// TIA Portal project "2022.10.18_视觉功能块（FB）" (V17)

(* hardware
DEVICE "S7-1200 station_1"  S7-1200 Station
   slot 0: "Rack_0"  S7-1200 Rack  Rack  V1.0
   slot 1: "PLC_1"  CPU 1215C DC/DC/Rly  6ES7 215-1HG40-0XB0  V4.5
*)

// ===== PLC "PLC_1"  CPU 1215C DC/DC/Rly =====

VAR_GLOBAL   // PLC tag table "默认变量表"
   "生成随机数" AT %M10.0 : Bool;
   "Tag_1" AT %M10.1 : Bool;
   "Tag_2" AT %M10.2 : Bool;
END_VAR

DATA_BLOCK "队列操作_DB"   // DB1
{ S7_Optimized_Access := 'TRUE' }
VERSION : 0.1
// stored: InstanceOfName 队列操作
"队列操作"
BEGIN
END_DATA_BLOCK

FUNCTION_BLOCK "队列操作"   // FB1, LAD
{ S7_Optimized_Access := 'TRUE' }
VERSION : 0.1
   VAR_INPUT
      生成随机数 : Bool;
      写入队列 : Bool;
      踢出队列 : Bool;
   END_VAR
   VAR_OUTPUT
      待加入队列的值 : UDInt;
      待踢出的数值 : UDInt;
   END_VAR
   VAR
      队列数据 : Array[1..10] of UDInt;
      数据暂存区 : Array[1..10] of UDInt;
      上一个RLO值1 : Bool;
      上一个RLO值2 : Bool;
      上一个RLO值3 : Bool;
      INDEX : DInt;
      RET_VAL : Int;
      系统时间 : DTL;
   END_VAR
   VAR_TEMP   // added for the SCL form of the ladder/FBD networks
      _w1 : Bool;
   END_VAR
BEGIN

REGION Network 1: 生成一个随机数
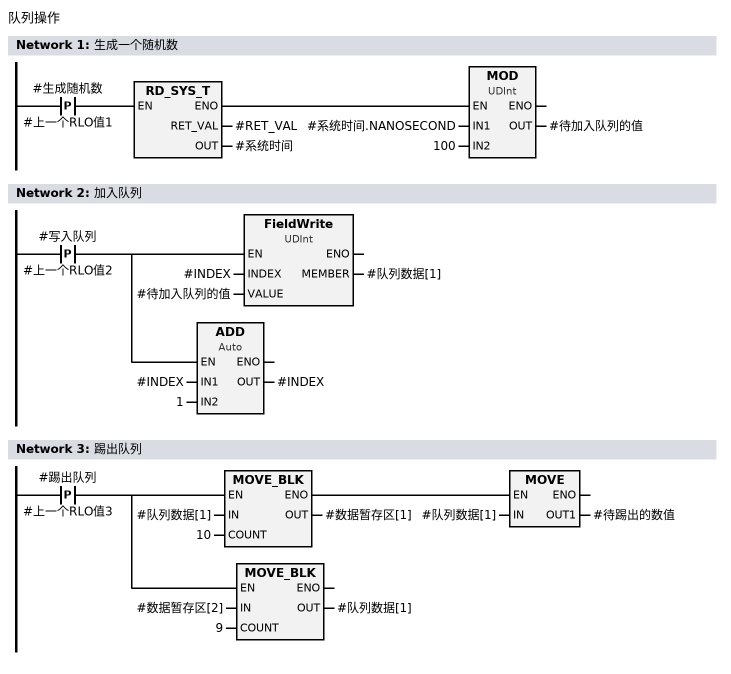
   // ENO of a box is taken as its EN; it also drops when the box reports an error
   #_w1 := #生成随机数 AND NOT #上一个RLO值1;   // rising edge of #生成随机数
   #上一个RLO值1 := #生成随机数;
   IF #_w1 THEN
       #RET_VAL := RD_SYS_T(OUT => #系统时间);
       #待加入队列的值 := #系统时间.NANOSECOND MOD 100;
   END_IF;
END_REGION

REGION Network 2: 加入队列
   // no SCL statement known for FieldWrite: written as a call
   #_w1 := #写入队列 AND NOT #上一个RLO值2;   // rising edge of #写入队列
   #上一个RLO值2 := #写入队列;
   IF #_w1 THEN
       FieldWrite(index := #INDEX, value := #待加入队列的值, member => #队列数据[1]);
       #INDEX := #INDEX + 1;
   END_IF;
END_REGION

REGION Network 3: 踢出队列
   #_w1 := #踢出队列 AND NOT #上一个RLO值3;   // rising edge of #踢出队列
   #上一个RLO值3 := #踢出队列;
   IF #_w1 THEN
       MOVE_BLK(IN := #队列数据[1], COUNT := 10, OUT => #数据暂存区[1]);
       #待踢出的数值 := #队列数据[1];
       MOVE_BLK(IN := #数据暂存区[2], COUNT := 9, OUT => #队列数据[1]);
   END_IF;
END_REGION
END_FUNCTION_BLOCK

ORGANIZATION_BLOCK "Main"   // OB1, LAD, ProgramCycle
TITLE = "Main Program Sweep (Cycle)"
{ S7_Optimized_Access := 'TRUE' }
VERSION : 0.1
   VAR_INPUT
      Initial_Call : Bool;   // Initial call of this OB
      Remanence : Bool;   // =True, if remanent data are available
   END_VAR
BEGIN

REGION Network 1
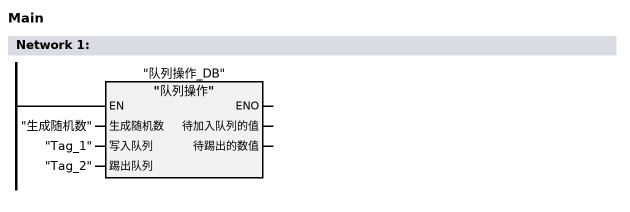
   RUNG wire#powerrail
      "队列操作_DB"(生成随机数 := "生成随机数", 写入队列 := "Tag_1", 踢出队列 := "Tag_2", 待加入队列的值 =>, 待踢出的数值 =>)
   END_RUNG
   // the same network as SCL:
   "队列操作_DB"(生成随机数 := "生成随机数", 写入队列 := "Tag_1", 踢出队列 := "Tag_2");   // "队列操作"
END_REGION
END_ORGANIZATION_BLOCK